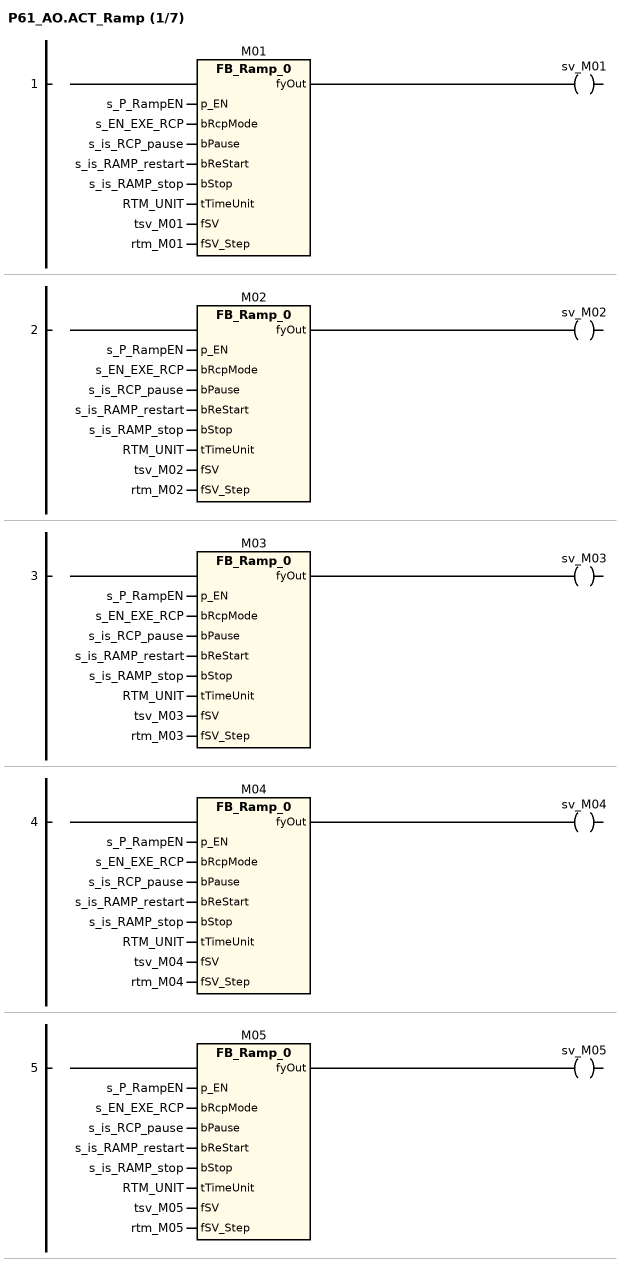
// NETWORK 1
M01(
    p_EN := s_P_RampEN,
    bRcpMode := s_EN_EXE_RCP,
    bPause := s_is_RCP_pause,
    bReStart := s_is_RAMP_restart,
    bStop := s_is_RAMP_stop,
    tTimeUnit := RTM_UNIT,
    fSV := tsv_M01,
    fSV_Step := rtm_M01); // FB_Ramp_0
sv_M01 := M01.fyOut;

// NETWORK 2
M02(
    p_EN := s_P_RampEN,
    bRcpMode := s_EN_EXE_RCP,
    bPause := s_is_RCP_pause,
    bReStart := s_is_RAMP_restart,
    bStop := s_is_RAMP_stop,
    tTimeUnit := RTM_UNIT,
    fSV := tsv_M02,
    fSV_Step := rtm_M02); // FB_Ramp_0
sv_M02 := M02.fyOut;

// NETWORK 3
M03(
    p_EN := s_P_RampEN,
    bRcpMode := s_EN_EXE_RCP,
    bPause := s_is_RCP_pause,
    bReStart := s_is_RAMP_restart,
    bStop := s_is_RAMP_stop,
    tTimeUnit := RTM_UNIT,
    fSV := tsv_M03,
    fSV_Step := rtm_M03); // FB_Ramp_0
sv_M03 := M03.fyOut;

// NETWORK 4
M04(
    p_EN := s_P_RampEN,
    bRcpMode := s_EN_EXE_RCP,
    bPause := s_is_RCP_pause,
    bReStart := s_is_RAMP_restart,
    bStop := s_is_RAMP_stop,
    tTimeUnit := RTM_UNIT,
    fSV := tsv_M04,
    fSV_Step := rtm_M04); // FB_Ramp_0
sv_M04 := M04.fyOut;

// NETWORK 5
M05(
    p_EN := s_P_RampEN,
    bRcpMode := s_EN_EXE_RCP,
    bPause := s_is_RCP_pause,
    bReStart := s_is_RAMP_restart,
    bStop := s_is_RAMP_stop,
    tTimeUnit := RTM_UNIT,
    fSV := tsv_M05,
    fSV_Step := rtm_M05); // FB_Ramp_0
sv_M05 := M05.fyOut;

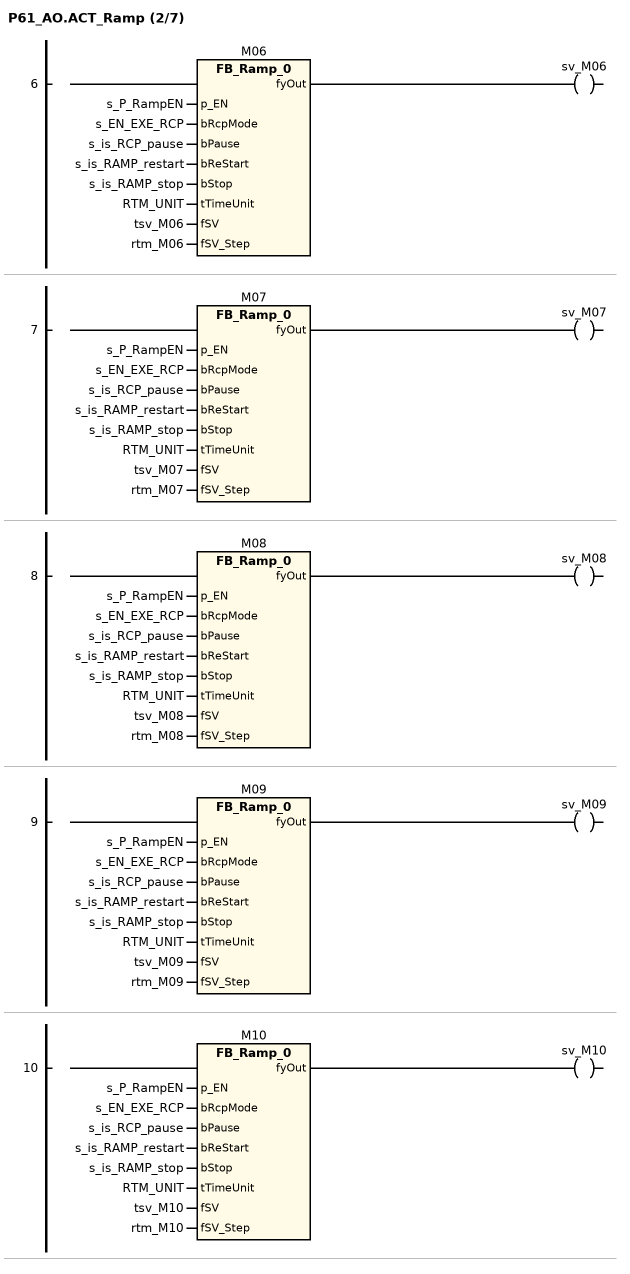
// NETWORK 6
M06(
    p_EN := s_P_RampEN,
    bRcpMode := s_EN_EXE_RCP,
    bPause := s_is_RCP_pause,
    bReStart := s_is_RAMP_restart,
    bStop := s_is_RAMP_stop,
    tTimeUnit := RTM_UNIT,
    fSV := tsv_M06,
    fSV_Step := rtm_M06); // FB_Ramp_0
sv_M06 := M06.fyOut;

// NETWORK 7
M07(
    p_EN := s_P_RampEN,
    bRcpMode := s_EN_EXE_RCP,
    bPause := s_is_RCP_pause,
    bReStart := s_is_RAMP_restart,
    bStop := s_is_RAMP_stop,
    tTimeUnit := RTM_UNIT,
    fSV := tsv_M07,
    fSV_Step := rtm_M07); // FB_Ramp_0
sv_M07 := M07.fyOut;

// NETWORK 8
M08(
    p_EN := s_P_RampEN,
    bRcpMode := s_EN_EXE_RCP,
    bPause := s_is_RCP_pause,
    bReStart := s_is_RAMP_restart,
    bStop := s_is_RAMP_stop,
    tTimeUnit := RTM_UNIT,
    fSV := tsv_M08,
    fSV_Step := rtm_M08); // FB_Ramp_0
sv_M08 := M08.fyOut;

// NETWORK 9
M09(
    p_EN := s_P_RampEN,
    bRcpMode := s_EN_EXE_RCP,
    bPause := s_is_RCP_pause,
    bReStart := s_is_RAMP_restart,
    bStop := s_is_RAMP_stop,
    tTimeUnit := RTM_UNIT,
    fSV := tsv_M09,
    fSV_Step := rtm_M09); // FB_Ramp_0
sv_M09 := M09.fyOut;

// NETWORK 10
M10(
    p_EN := s_P_RampEN,
    bRcpMode := s_EN_EXE_RCP,
    bPause := s_is_RCP_pause,
    bReStart := s_is_RAMP_restart,
    bStop := s_is_RAMP_stop,
    tTimeUnit := RTM_UNIT,
    fSV := tsv_M10,
    fSV_Step := rtm_M10); // FB_Ramp_0
sv_M10 := M10.fyOut;

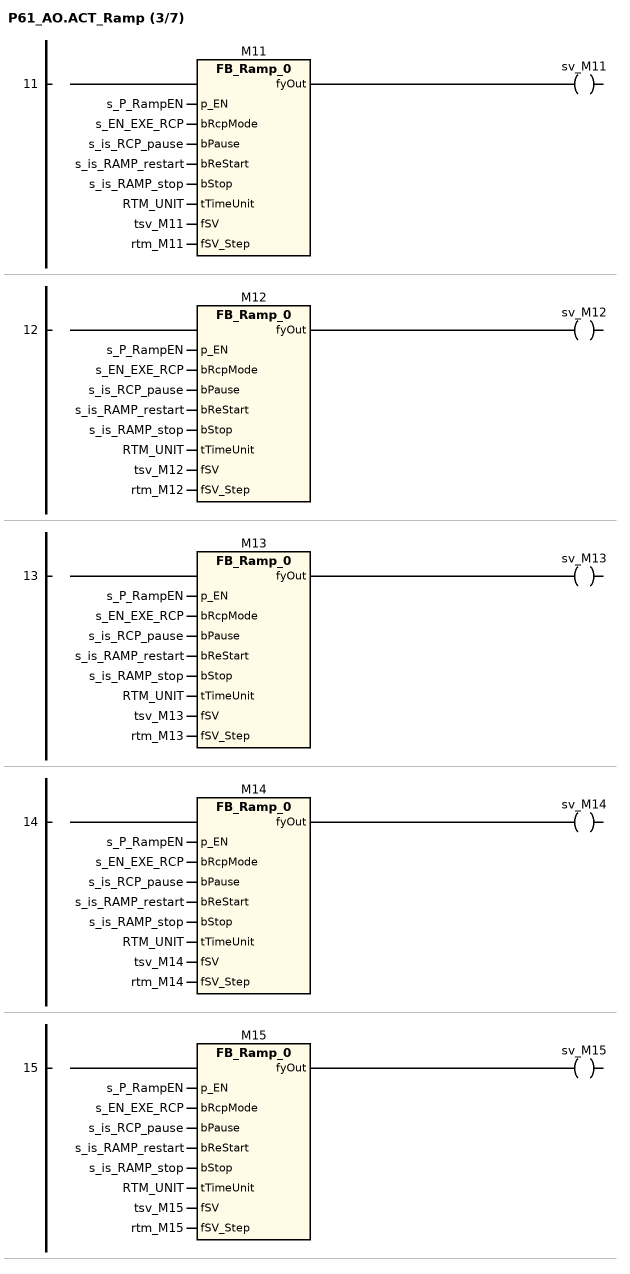
// NETWORK 11
M11(
    p_EN := s_P_RampEN,
    bRcpMode := s_EN_EXE_RCP,
    bPause := s_is_RCP_pause,
    bReStart := s_is_RAMP_restart,
    bStop := s_is_RAMP_stop,
    tTimeUnit := RTM_UNIT,
    fSV := tsv_M11,
    fSV_Step := rtm_M11); // FB_Ramp_0
sv_M11 := M11.fyOut;

// NETWORK 12
M12(
    p_EN := s_P_RampEN,
    bRcpMode := s_EN_EXE_RCP,
    bPause := s_is_RCP_pause,
    bReStart := s_is_RAMP_restart,
    bStop := s_is_RAMP_stop,
    tTimeUnit := RTM_UNIT,
    fSV := tsv_M12,
    fSV_Step := rtm_M12); // FB_Ramp_0
sv_M12 := M12.fyOut;

// NETWORK 13
M13(
    p_EN := s_P_RampEN,
    bRcpMode := s_EN_EXE_RCP,
    bPause := s_is_RCP_pause,
    bReStart := s_is_RAMP_restart,
    bStop := s_is_RAMP_stop,
    tTimeUnit := RTM_UNIT,
    fSV := tsv_M13,
    fSV_Step := rtm_M13); // FB_Ramp_0
sv_M13 := M13.fyOut;

// NETWORK 14
M14(
    p_EN := s_P_RampEN,
    bRcpMode := s_EN_EXE_RCP,
    bPause := s_is_RCP_pause,
    bReStart := s_is_RAMP_restart,
    bStop := s_is_RAMP_stop,
    tTimeUnit := RTM_UNIT,
    fSV := tsv_M14,
    fSV_Step := rtm_M14); // FB_Ramp_0
sv_M14 := M14.fyOut;

// NETWORK 15
M15(
    p_EN := s_P_RampEN,
    bRcpMode := s_EN_EXE_RCP,
    bPause := s_is_RCP_pause,
    bReStart := s_is_RAMP_restart,
    bStop := s_is_RAMP_stop,
    tTimeUnit := RTM_UNIT,
    fSV := tsv_M15,
    fSV_Step := rtm_M15); // FB_Ramp_0
sv_M15 := M15.fyOut;

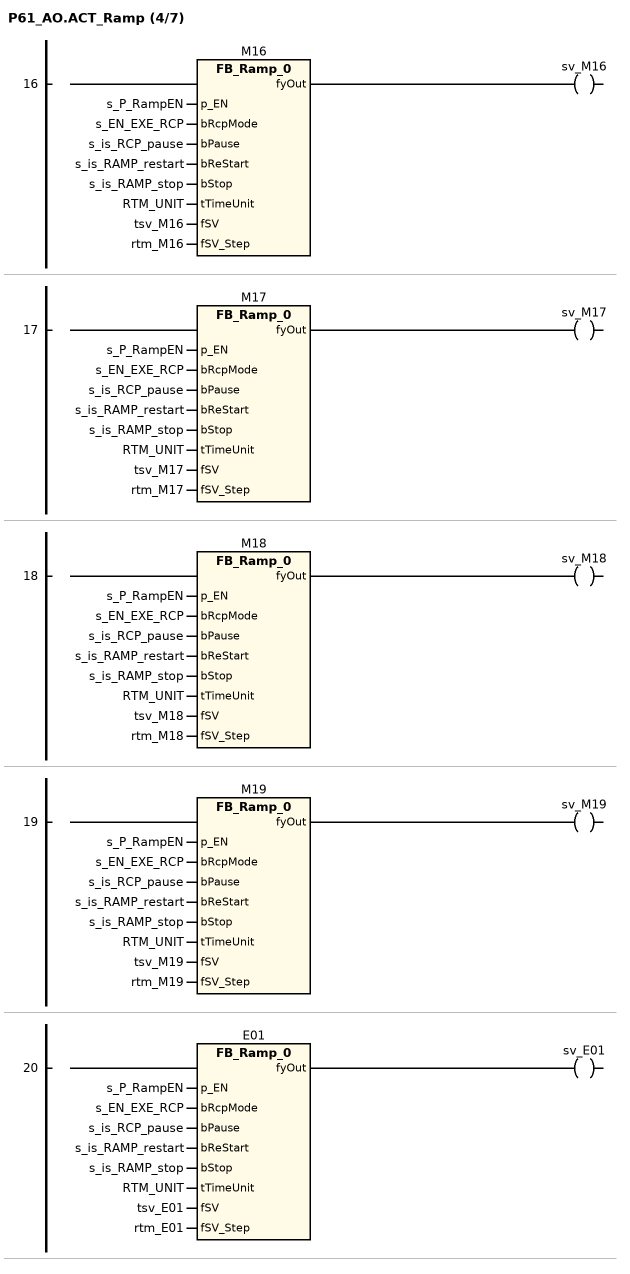
// NETWORK 16
M16(
    p_EN := s_P_RampEN,
    bRcpMode := s_EN_EXE_RCP,
    bPause := s_is_RCP_pause,
    bReStart := s_is_RAMP_restart,
    bStop := s_is_RAMP_stop,
    tTimeUnit := RTM_UNIT,
    fSV := tsv_M16,
    fSV_Step := rtm_M16); // FB_Ramp_0
sv_M16 := M16.fyOut;

// NETWORK 17
M17(
    p_EN := s_P_RampEN,
    bRcpMode := s_EN_EXE_RCP,
    bPause := s_is_RCP_pause,
    bReStart := s_is_RAMP_restart,
    bStop := s_is_RAMP_stop,
    tTimeUnit := RTM_UNIT,
    fSV := tsv_M17,
    fSV_Step := rtm_M17); // FB_Ramp_0
sv_M17 := M17.fyOut;

// NETWORK 18
M18(
    p_EN := s_P_RampEN,
    bRcpMode := s_EN_EXE_RCP,
    bPause := s_is_RCP_pause,
    bReStart := s_is_RAMP_restart,
    bStop := s_is_RAMP_stop,
    tTimeUnit := RTM_UNIT,
    fSV := tsv_M18,
    fSV_Step := rtm_M18); // FB_Ramp_0
sv_M18 := M18.fyOut;

// NETWORK 19
M19(
    p_EN := s_P_RampEN,
    bRcpMode := s_EN_EXE_RCP,
    bPause := s_is_RCP_pause,
    bReStart := s_is_RAMP_restart,
    bStop := s_is_RAMP_stop,
    tTimeUnit := RTM_UNIT,
    fSV := tsv_M19,
    fSV_Step := rtm_M19); // FB_Ramp_0
sv_M19 := M19.fyOut;

// NETWORK 20
E01(
    p_EN := s_P_RampEN,
    bRcpMode := s_EN_EXE_RCP,
    bPause := s_is_RCP_pause,
    bReStart := s_is_RAMP_restart,
    bStop := s_is_RAMP_stop,
    tTimeUnit := RTM_UNIT,
    fSV := tsv_E01,
    fSV_Step := rtm_E01); // FB_Ramp_0
sv_E01 := E01.fyOut;

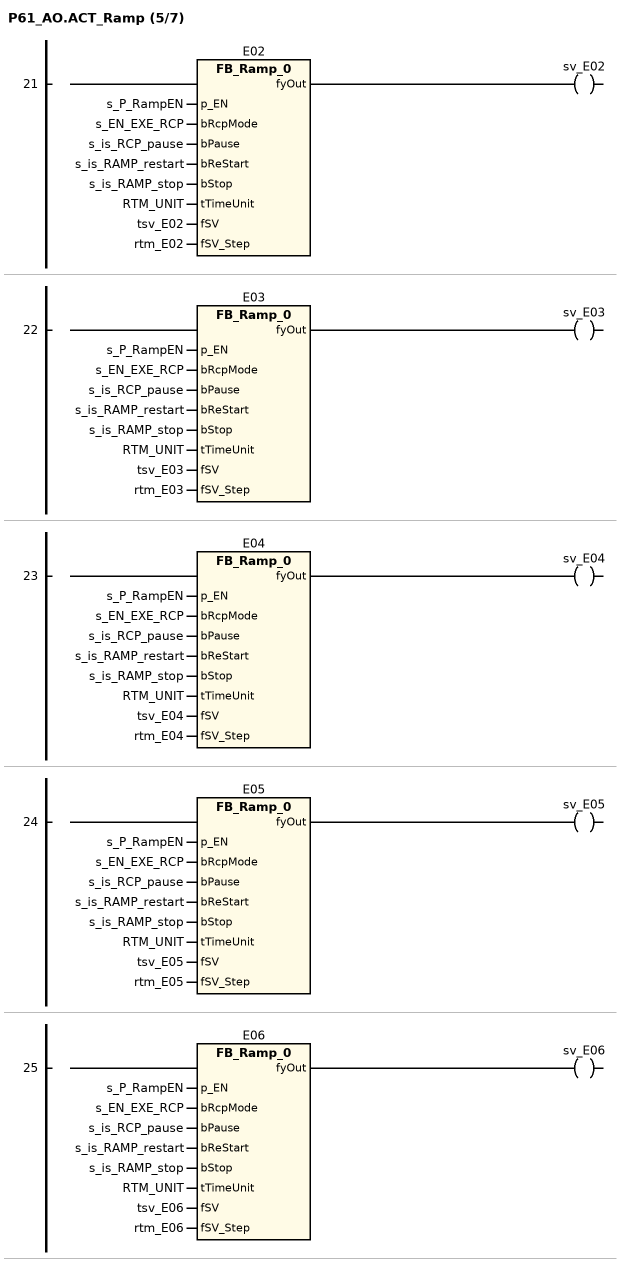
// NETWORK 21
E02(
    p_EN := s_P_RampEN,
    bRcpMode := s_EN_EXE_RCP,
    bPause := s_is_RCP_pause,
    bReStart := s_is_RAMP_restart,
    bStop := s_is_RAMP_stop,
    tTimeUnit := RTM_UNIT,
    fSV := tsv_E02,
    fSV_Step := rtm_E02); // FB_Ramp_0
sv_E02 := E02.fyOut;

// NETWORK 22
E03(
    p_EN := s_P_RampEN,
    bRcpMode := s_EN_EXE_RCP,
    bPause := s_is_RCP_pause,
    bReStart := s_is_RAMP_restart,
    bStop := s_is_RAMP_stop,
    tTimeUnit := RTM_UNIT,
    fSV := tsv_E03,
    fSV_Step := rtm_E03); // FB_Ramp_0
sv_E03 := E03.fyOut;

// NETWORK 23
E04(
    p_EN := s_P_RampEN,
    bRcpMode := s_EN_EXE_RCP,
    bPause := s_is_RCP_pause,
    bReStart := s_is_RAMP_restart,
    bStop := s_is_RAMP_stop,
    tTimeUnit := RTM_UNIT,
    fSV := tsv_E04,
    fSV_Step := rtm_E04); // FB_Ramp_0
sv_E04 := E04.fyOut;

// NETWORK 24
E05(
    p_EN := s_P_RampEN,
    bRcpMode := s_EN_EXE_RCP,
    bPause := s_is_RCP_pause,
    bReStart := s_is_RAMP_restart,
    bStop := s_is_RAMP_stop,
    tTimeUnit := RTM_UNIT,
    fSV := tsv_E05,
    fSV_Step := rtm_E05); // FB_Ramp_0
sv_E05 := E05.fyOut;

// NETWORK 25
E06(
    p_EN := s_P_RampEN,
    bRcpMode := s_EN_EXE_RCP,
    bPause := s_is_RCP_pause,
    bReStart := s_is_RAMP_restart,
    bStop := s_is_RAMP_stop,
    tTimeUnit := RTM_UNIT,
    fSV := tsv_E06,
    fSV_Step := rtm_E06); // FB_Ramp_0
sv_E06 := E06.fyOut;

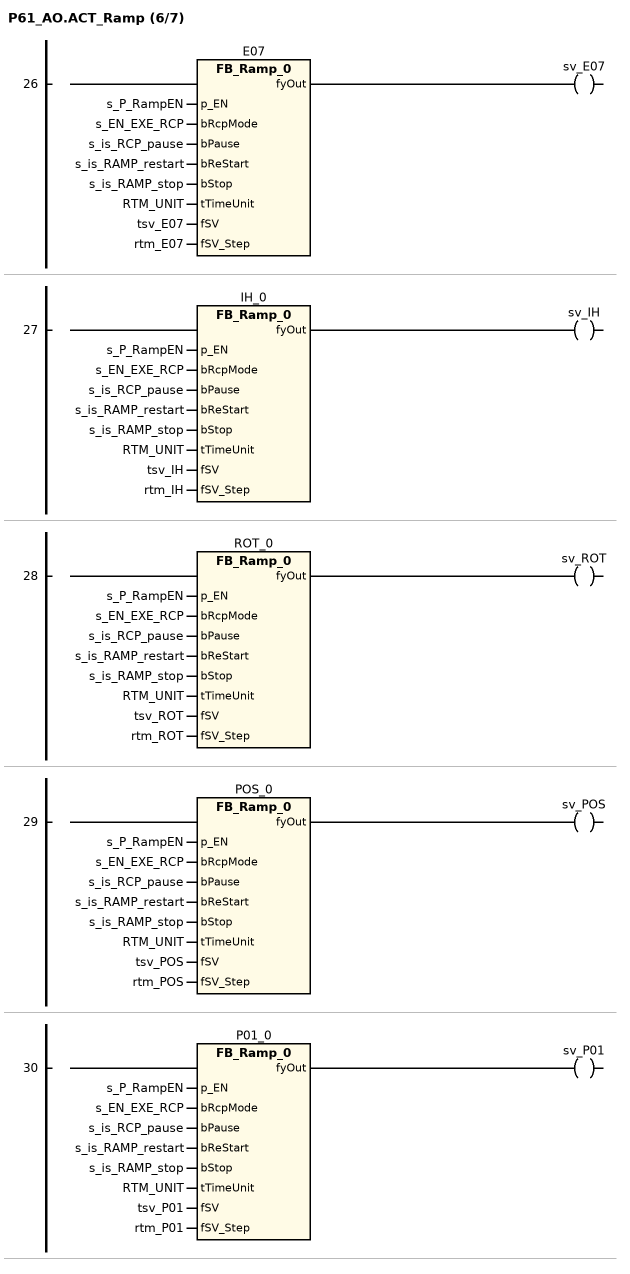
// NETWORK 26
E07(
    p_EN := s_P_RampEN,
    bRcpMode := s_EN_EXE_RCP,
    bPause := s_is_RCP_pause,
    bReStart := s_is_RAMP_restart,
    bStop := s_is_RAMP_stop,
    tTimeUnit := RTM_UNIT,
    fSV := tsv_E07,
    fSV_Step := rtm_E07); // FB_Ramp_0
sv_E07 := E07.fyOut;

// NETWORK 27
IH_0(
    p_EN := s_P_RampEN,
    bRcpMode := s_EN_EXE_RCP,
    bPause := s_is_RCP_pause,
    bReStart := s_is_RAMP_restart,
    bStop := s_is_RAMP_stop,
    tTimeUnit := RTM_UNIT,
    fSV := tsv_IH,
    fSV_Step := rtm_IH); // FB_Ramp_0
sv_IH := IH_0.fyOut;

// NETWORK 28
ROT_0(
    p_EN := s_P_RampEN,
    bRcpMode := s_EN_EXE_RCP,
    bPause := s_is_RCP_pause,
    bReStart := s_is_RAMP_restart,
    bStop := s_is_RAMP_stop,
    tTimeUnit := RTM_UNIT,
    fSV := tsv_ROT,
    fSV_Step := rtm_ROT); // FB_Ramp_0
sv_ROT := ROT_0.fyOut;

// NETWORK 29
POS_0(
    p_EN := s_P_RampEN,
    bRcpMode := s_EN_EXE_RCP,
    bPause := s_is_RCP_pause,
    bReStart := s_is_RAMP_restart,
    bStop := s_is_RAMP_stop,
    tTimeUnit := RTM_UNIT,
    fSV := tsv_POS,
    fSV_Step := rtm_POS); // FB_Ramp_0
sv_POS := POS_0.fyOut;

// NETWORK 30
P01_0(
    p_EN := s_P_RampEN,
    bRcpMode := s_EN_EXE_RCP,
    bPause := s_is_RCP_pause,
    bReStart := s_is_RAMP_restart,
    bStop := s_is_RAMP_stop,
    tTimeUnit := RTM_UNIT,
    fSV := tsv_P01,
    fSV_Step := rtm_P01); // FB_Ramp_0
sv_P01 := P01_0.fyOut;

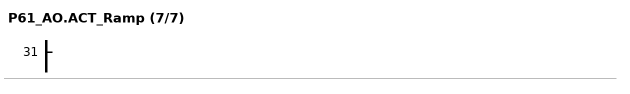
// NETWORK 31
END_ACTION

ACTION ACT_Ramp_OLD:
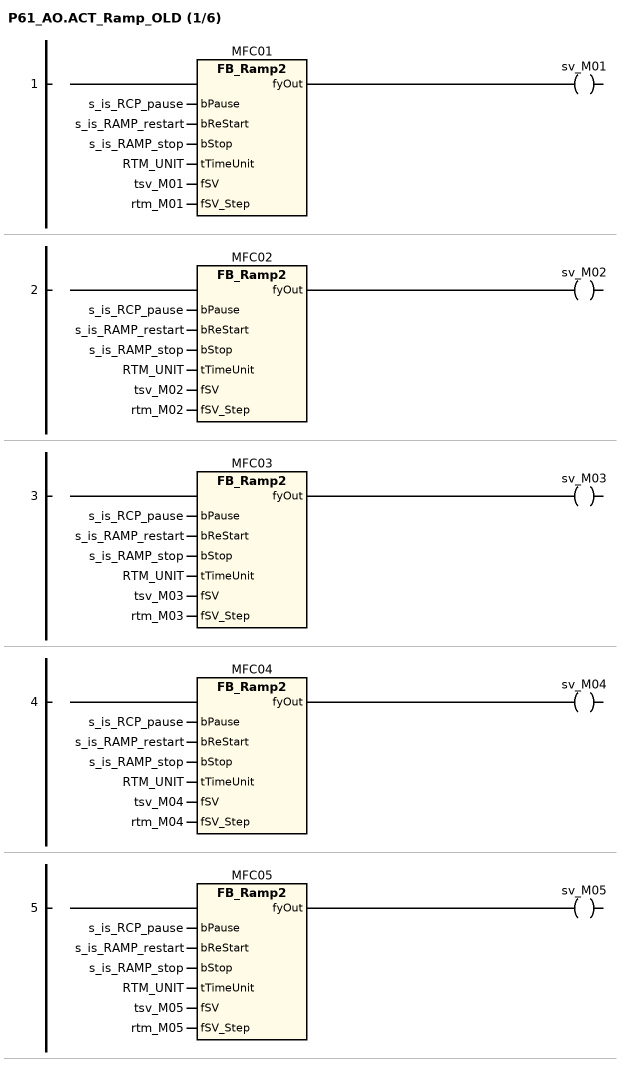
// NETWORK 1
MFC01(
    bPause := s_is_RCP_pause,
    bReStart := s_is_RAMP_restart,
    bStop := s_is_RAMP_stop,
    tTimeUnit := RTM_UNIT,
    fSV := tsv_M01,
    fSV_Step := rtm_M01); // FB_Ramp2
sv_M01 := MFC01.fyOut;

// NETWORK 2
MFC02(
    bPause := s_is_RCP_pause,
    bReStart := s_is_RAMP_restart,
    bStop := s_is_RAMP_stop,
    tTimeUnit := RTM_UNIT,
    fSV := tsv_M02,
    fSV_Step := rtm_M02); // FB_Ramp2
sv_M02 := MFC02.fyOut;

// NETWORK 3
MFC03(
    bPause := s_is_RCP_pause,
    bReStart := s_is_RAMP_restart,
    bStop := s_is_RAMP_stop,
    tTimeUnit := RTM_UNIT,
    fSV := tsv_M03,
    fSV_Step := rtm_M03); // FB_Ramp2
sv_M03 := MFC03.fyOut;

// NETWORK 4
MFC04(
    bPause := s_is_RCP_pause,
    bReStart := s_is_RAMP_restart,
    bStop := s_is_RAMP_stop,
    tTimeUnit := RTM_UNIT,
    fSV := tsv_M04,
    fSV_Step := rtm_M04); // FB_Ramp2
sv_M04 := MFC04.fyOut;

// NETWORK 5
MFC05(
    bPause := s_is_RCP_pause,
    bReStart := s_is_RAMP_restart,
    bStop := s_is_RAMP_stop,
    tTimeUnit := RTM_UNIT,
    fSV := tsv_M05,
    fSV_Step := rtm_M05); // FB_Ramp2
sv_M05 := MFC05.fyOut;

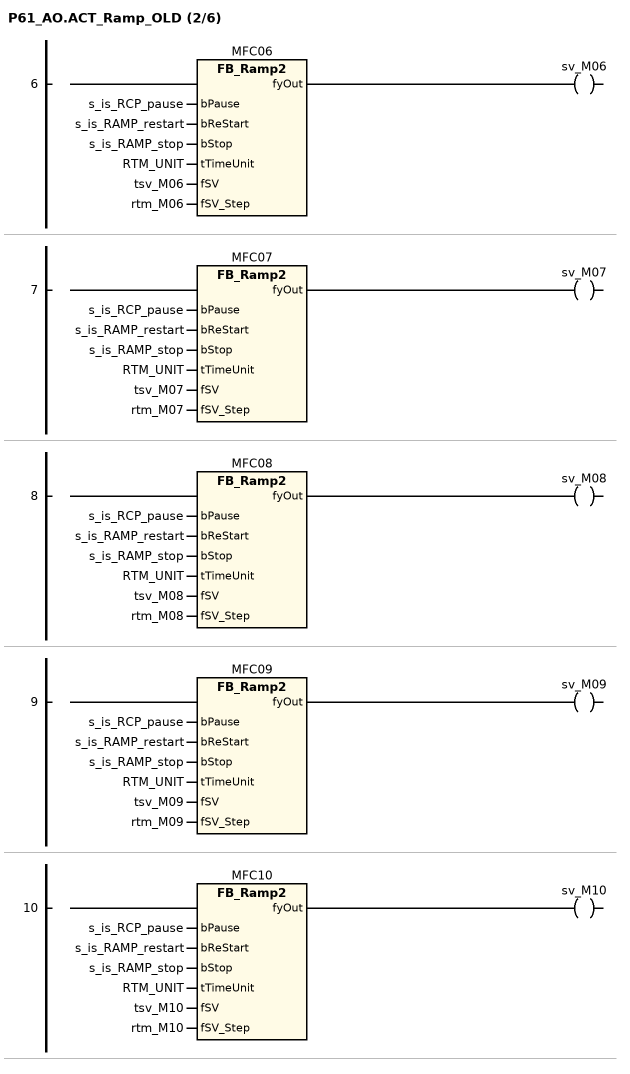
// NETWORK 6
MFC06(
    bPause := s_is_RCP_pause,
    bReStart := s_is_RAMP_restart,
    bStop := s_is_RAMP_stop,
    tTimeUnit := RTM_UNIT,
    fSV := tsv_M06,
    fSV_Step := rtm_M06); // FB_Ramp2
sv_M06 := MFC06.fyOut;

// NETWORK 7
MFC07(
    bPause := s_is_RCP_pause,
    bReStart := s_is_RAMP_restart,
    bStop := s_is_RAMP_stop,
    tTimeUnit := RTM_UNIT,
    fSV := tsv_M07,
    fSV_Step := rtm_M07); // FB_Ramp2
sv_M07 := MFC07.fyOut;

// NETWORK 8
MFC08(
    bPause := s_is_RCP_pause,
    bReStart := s_is_RAMP_restart,
    bStop := s_is_RAMP_stop,
    tTimeUnit := RTM_UNIT,
    fSV := tsv_M08,
    fSV_Step := rtm_M08); // FB_Ramp2
sv_M08 := MFC08.fyOut;

// NETWORK 9
MFC09(
    bPause := s_is_RCP_pause,
    bReStart := s_is_RAMP_restart,
    bStop := s_is_RAMP_stop,
    tTimeUnit := RTM_UNIT,
    fSV := tsv_M09,
    fSV_Step := rtm_M09); // FB_Ramp2
sv_M09 := MFC09.fyOut;

// NETWORK 10
MFC10(
    bPause := s_is_RCP_pause,
    bReStart := s_is_RAMP_restart,
    bStop := s_is_RAMP_stop,
    tTimeUnit := RTM_UNIT,
    fSV := tsv_M10,
    fSV_Step := rtm_M10); // FB_Ramp2
sv_M10 := MFC10.fyOut;

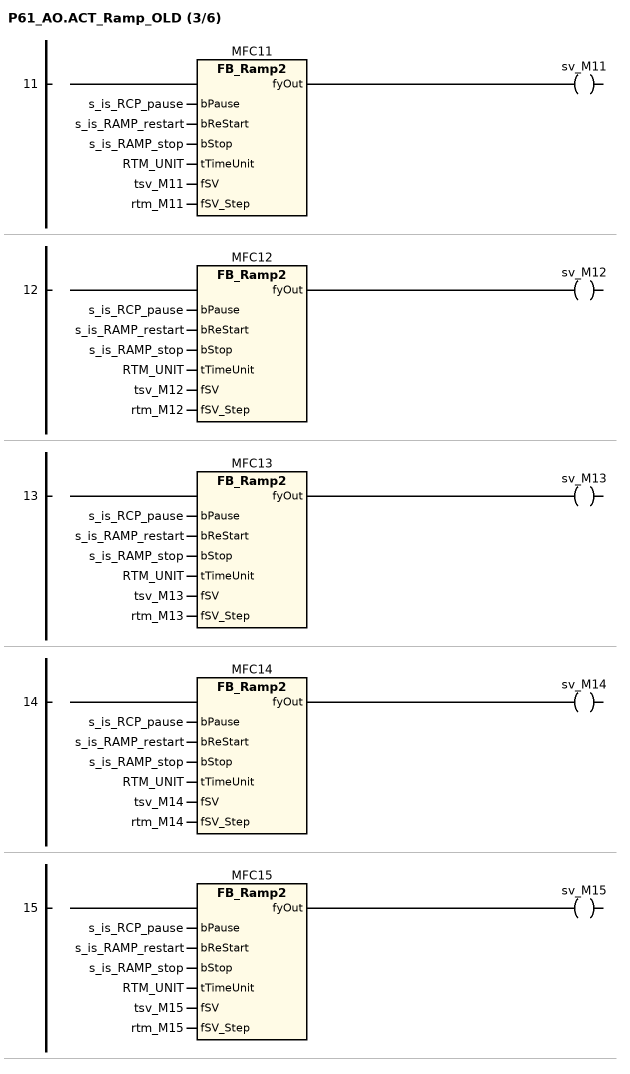
// NETWORK 11
MFC11(
    bPause := s_is_RCP_pause,
    bReStart := s_is_RAMP_restart,
    bStop := s_is_RAMP_stop,
    tTimeUnit := RTM_UNIT,
    fSV := tsv_M11,
    fSV_Step := rtm_M11); // FB_Ramp2
sv_M11 := MFC11.fyOut;

// NETWORK 12
MFC12(
    bPause := s_is_RCP_pause,
    bReStart := s_is_RAMP_restart,
    bStop := s_is_RAMP_stop,
    tTimeUnit := RTM_UNIT,
    fSV := tsv_M12,
    fSV_Step := rtm_M12); // FB_Ramp2
sv_M12 := MFC12.fyOut;

// NETWORK 13
MFC13(
    bPause := s_is_RCP_pause,
    bReStart := s_is_RAMP_restart,
    bStop := s_is_RAMP_stop,
    tTimeUnit := RTM_UNIT,
    fSV := tsv_M13,
    fSV_Step := rtm_M13); // FB_Ramp2
sv_M13 := MFC13.fyOut;

// NETWORK 14
MFC14(
    bPause := s_is_RCP_pause,
    bReStart := s_is_RAMP_restart,
    bStop := s_is_RAMP_stop,
    tTimeUnit := RTM_UNIT,
    fSV := tsv_M14,
    fSV_Step := rtm_M14); // FB_Ramp2
sv_M14 := MFC14.fyOut;

// NETWORK 15
MFC15(
    bPause := s_is_RCP_pause,
    bReStart := s_is_RAMP_restart,
    bStop := s_is_RAMP_stop,
    tTimeUnit := RTM_UNIT,
    fSV := tsv_M15,
    fSV_Step := rtm_M15); // FB_Ramp2
sv_M15 := MFC15.fyOut;

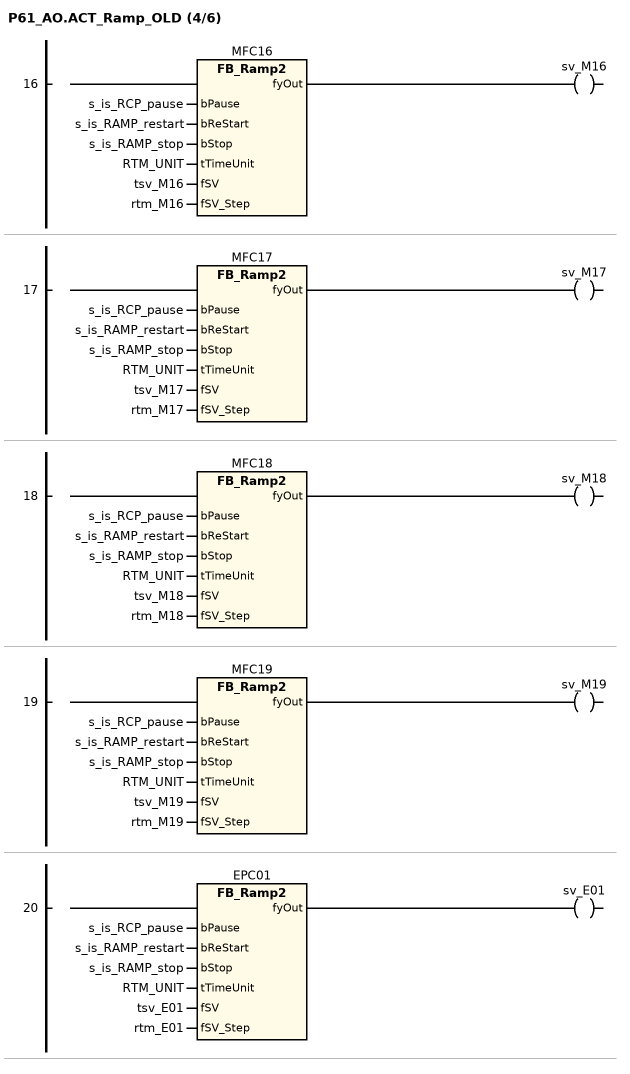
// NETWORK 16
MFC16(
    bPause := s_is_RCP_pause,
    bReStart := s_is_RAMP_restart,
    bStop := s_is_RAMP_stop,
    tTimeUnit := RTM_UNIT,
    fSV := tsv_M16,
    fSV_Step := rtm_M16); // FB_Ramp2
sv_M16 := MFC16.fyOut;

// NETWORK 17
MFC17(
    bPause := s_is_RCP_pause,
    bReStart := s_is_RAMP_restart,
    bStop := s_is_RAMP_stop,
    tTimeUnit := RTM_UNIT,
    fSV := tsv_M17,
    fSV_Step := rtm_M17); // FB_Ramp2
sv_M17 := MFC17.fyOut;

// NETWORK 18
MFC18(
    bPause := s_is_RCP_pause,
    bReStart := s_is_RAMP_restart,
    bStop := s_is_RAMP_stop,
    tTimeUnit := RTM_UNIT,
    fSV := tsv_M18,
    fSV_Step := rtm_M18); // FB_Ramp2
sv_M18 := MFC18.fyOut;

// NETWORK 19
MFC19(
    bPause := s_is_RCP_pause,
    bReStart := s_is_RAMP_restart,
    bStop := s_is_RAMP_stop,
    tTimeUnit := RTM_UNIT,
    fSV := tsv_M19,
    fSV_Step := rtm_M19); // FB_Ramp2
sv_M19 := MFC19.fyOut;

// NETWORK 20
EPC01(
    bPause := s_is_RCP_pause,
    bReStart := s_is_RAMP_restart,
    bStop := s_is_RAMP_stop,
    tTimeUnit := RTM_UNIT,
    fSV := tsv_E01,
    fSV_Step := rtm_E01); // FB_Ramp2
sv_E01 := EPC01.fyOut;

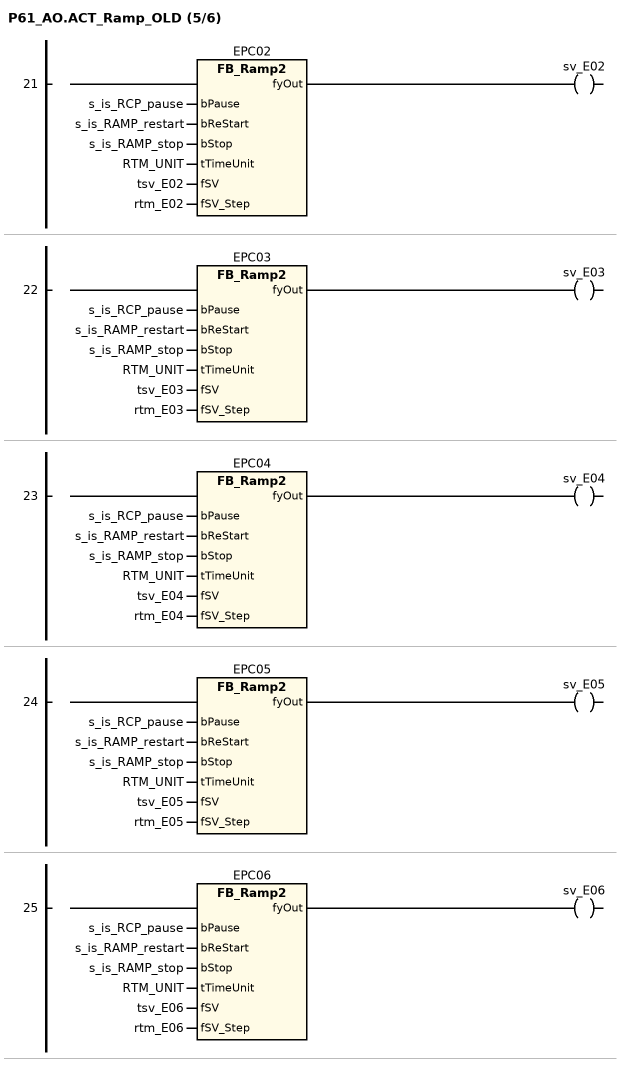
// NETWORK 21
EPC02(
    bPause := s_is_RCP_pause,
    bReStart := s_is_RAMP_restart,
    bStop := s_is_RAMP_stop,
    tTimeUnit := RTM_UNIT,
    fSV := tsv_E02,
    fSV_Step := rtm_E02); // FB_Ramp2
sv_E02 := EPC02.fyOut;

// NETWORK 22
EPC03(
    bPause := s_is_RCP_pause,
    bReStart := s_is_RAMP_restart,
    bStop := s_is_RAMP_stop,
    tTimeUnit := RTM_UNIT,
    fSV := tsv_E03,
    fSV_Step := rtm_E03); // FB_Ramp2
sv_E03 := EPC03.fyOut;

// NETWORK 23
EPC04(
    bPause := s_is_RCP_pause,
    bReStart := s_is_RAMP_restart,
    bStop := s_is_RAMP_stop,
    tTimeUnit := RTM_UNIT,
    fSV := tsv_E04,
    fSV_Step := rtm_E04); // FB_Ramp2
sv_E04 := EPC04.fyOut;

// NETWORK 24
EPC05(
    bPause := s_is_RCP_pause,
    bReStart := s_is_RAMP_restart,
    bStop := s_is_RAMP_stop,
    tTimeUnit := RTM_UNIT,
    fSV := tsv_E05,
    fSV_Step := rtm_E05); // FB_Ramp2
sv_E05 := EPC05.fyOut;

// NETWORK 25
EPC06(
    bPause := s_is_RCP_pause,
    bReStart := s_is_RAMP_restart,
    bStop := s_is_RAMP_stop,
    tTimeUnit := RTM_UNIT,
    fSV := tsv_E06,
    fSV_Step := rtm_E06); // FB_Ramp2
sv_E06 := EPC06.fyOut;

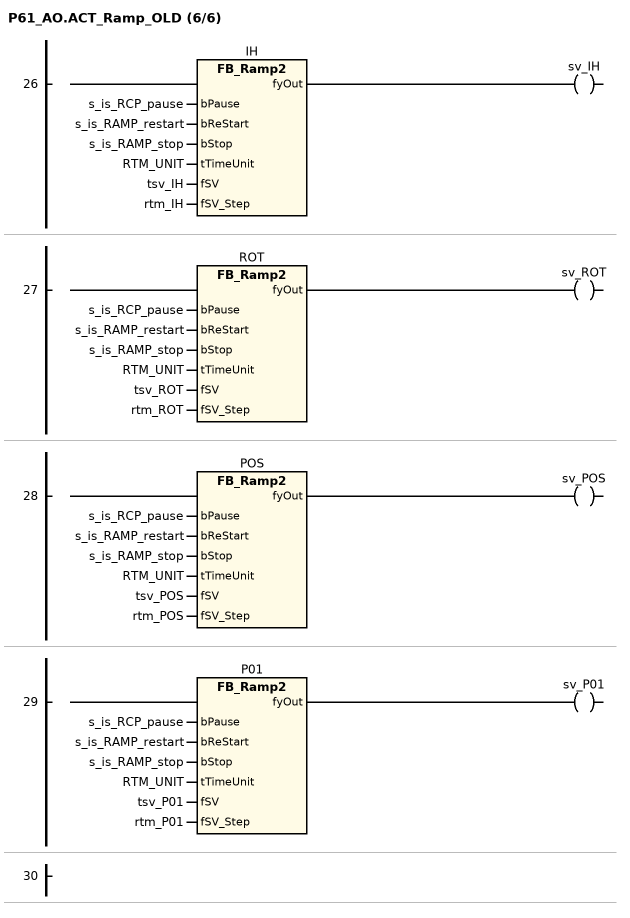
// NETWORK 26
IH(
    bPause := s_is_RCP_pause,
    bReStart := s_is_RAMP_restart,
    bStop := s_is_RAMP_stop,
    tTimeUnit := RTM_UNIT,
    fSV := tsv_IH,
    fSV_Step := rtm_IH); // FB_Ramp2
sv_IH := IH.fyOut;

// NETWORK 27
ROT(
    bPause := s_is_RCP_pause,
    bReStart := s_is_RAMP_restart,
    bStop := s_is_RAMP_stop,
    tTimeUnit := RTM_UNIT,
    fSV := tsv_ROT,
    fSV_Step := rtm_ROT); // FB_Ramp2
sv_ROT := ROT.fyOut;

// NETWORK 28
POS(
    bPause := s_is_RCP_pause,
    bReStart := s_is_RAMP_restart,
    bStop := s_is_RAMP_stop,
    tTimeUnit := RTM_UNIT,
    fSV := tsv_POS,
    fSV_Step := rtm_POS); // FB_Ramp2
sv_POS := POS.fyOut;

// NETWORK 29
P01(
    bPause := s_is_RCP_pause,
    bReStart := s_is_RAMP_restart,
    bStop := s_is_RAMP_stop,
    tTimeUnit := RTM_UNIT,
    fSV := tsv_P01,
    fSV_Step := rtm_P01); // FB_Ramp2
sv_P01 := P01.fyOut;

// NETWORK 30
END_ACTION

END_PROGRAM

// ---- POUs/MR_PRG/REF_P02_KL1501.TcPOU
PROGRAM REF_P02_KL1501
VAR
	//bError: BOOL;
	t_1S: TON;	
	
	iStatus: USINT;
	in1: UINT;
	in2: UINT;
		
	encCount: UDINT;
	inData: ST_KL1501InData;
	outData: ST_KL1501OutData;
	KL1501Cfg: FB_KL1501Config;
	
	One_Turn_PLS: REAL ;
	PLS_Old: REAL := 0;
	PLS_New: REAL := 0;
	PLS_Diff: REAL := 0;
	Encoder_Max: REAL := 4294967295; //UINT Range 0 ~ 65,535
	RPM_PV: REAL := 0;
	FB_RPM_AVG: FB_AVG10;
	RPM_AVG: REAL;
    BLDC_MAX_RPM_PLS: REAL := 36000;//genicom : 12PULSE * 3000RPM = 36,000PULSE, china hvpe :500PULSE * 4000RPM = 2,000,000PULSE	
END_VAR

t_1S(PT := T#1S);
t_1S.IN := ON;

//KL1501 Not Use
(*

inData.iState := XA_ENC_ST;
inData.arrDataIn[0] := XA_ENC_IN[0];
inData.arrDataIn[1] := XA_ENC_IN[1];

IF t_1S.Q THEN
	t_1S.IN := Off;
	
	ACT_KL1501();
	
	//Rotation - BLDC Encoder
	pv_ENC := PLS_New := UDINT_TO_REAL(encCount);
	IF N_MAX[29] > 0 THEN
		One_Turn_PLS := BLDC_MAX_RPM_PLS / N_MAX[29];
	ELSE
		One_Turn_PLS := 1;
	END_IF
	IF PLS_New <> PLS_Old THEN //pulse input check
		IF PLS_New <= PLS_Old THEN//Ring counter Check
			PLS_New := PLS_New + Encoder_Max;
		END_IF
		PLS_Diff := PLS_New - PLS_Old;//PLS_Diff is always + value	
		IF PLS_Diff >= 0 THEN	//PLS_Diff is sometime abnormal value
			pv_ROT_inchPulse := pv_ROT_inchPulse + PLS_Diff; //PLS_Diff is always + value
			pv_ROT_1turnPulse := pv_ROT_1turnPulse + PLS_Diff; //PLS_Diff is always + value
			RPM_PV := PLS_Diff * 60 / One_Turn_PLS ;// 60 = 60Sec
		END_IF
		pv_ROT := RPM_PV;
	ELSE	
		pv_ROT := 0;	
	END_IF
	
	IF pv_ROT_1turnPulse >= One_Turn_PLS THEN
		pv_ROT_1turnPulse := pv_ROT_1turnPulse - One_Turn_PLS;
	END_IF
	pv_ROT_DEGREE := pv_ROT_1turnPulse *  360 / One_Turn_PLS;
	
	is_ROT_plsActived := PLS_New <> PLS_Old;
	PLS_Old := PLS_New;	

END_IF;//end 1Sec Timer.Q

*)

ACTION ACT_KL1501:
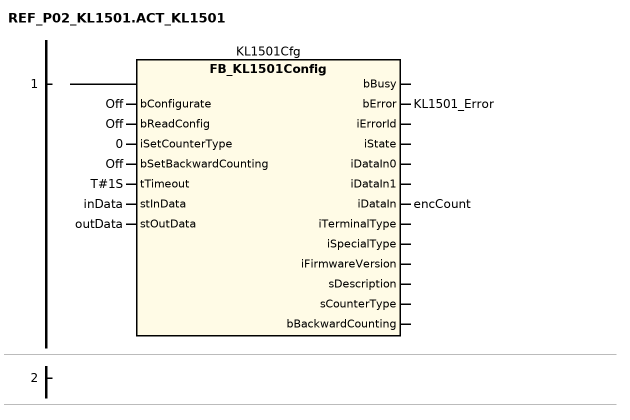
// NETWORK 1
KL1501Cfg(
    bConfigurate := Off,
    bReadConfig := Off,
    iSetCounterType := 0,
    bSetBackwardCounting := Off,
    tTimeout := T#1S,
    stInData := inData,
    stOutData := outData,
    bError => KL1501_Error,
    iDataIn => encCount); // FB_KL1501Config

// NETWORK 2
END_ACTION

END_PROGRAM

// ---- POUs/P02_P2P/P00_Task_Fast.TcPOU
PROGRAM P00_Task_Fast
VAR
END_VAR


Task_Fast_LH();
Task_Fast_TB();

END_PROGRAM

// ---- POUs/P02_P2P/Task_Fast_LH.TcPOU
PROGRAM Task_Fast_LH
VAR
	//LineHeater Controller(MC9-8RD0SS32) x 1EA
	(* background communication with the KL6031 terminal (22byte) *)
	fbCtrl: SerialLineControl;
	bCtrlError: BOOL;
	eCtrlErrorID: ComError_t;
	fbKLConfig: KL6configuration;
	bKLConfigError: BOOL;
	eKLConfigErrorID: ComError_t;
	bKLConfigExe: BOOL := TRUE;
END_VAR

//LH: Line Heater x 8EA -> 8Channel TIC 1EA
//Maker: HANYOUNG NUX
//Model: MC9-8RD0SS32
//Temp Range: -15 ~200℃
//RS485: 9600, DataBit(8), Parity(None), StopBit(1)
//BCC Check X
fbCtrl(
	Mode:= SERIALLINEMODE_KL6_22B_STANDARD,
	pComIn:= ADR(in22B_LH),
	pComOut:= ADR(out22B_LH),
	SizeComIn:= SIZEOF(in22B_LH),
	Error=> ,
	ErrorID=> ,
	TxBuffer:= TxBuf_LH,
	RxBuffer:= RxBuf_LH );
IF fbCtrl.Error THEN
	bCtrlError := TRUE;
	eCtrlErrorID := fbCtrl.ErrorID;
END_IF

END_PROGRAM

// ---- POUs/P02_P2P/Task_Fast_TB.TcPOU
PROGRAM Task_Fast_TB
VAR
	//Thermal Bath(HEBC002-WA10) x 6EA
	(* background communication with the KL6031 terminal (22byte) *)
	fbCtrl: SerialLineControl;
	bCtrlError: BOOL;
	eCtrlErrorID: ComError_t;
	fbKLConfig: KL6configuration;
	bKLConfigError: BOOL;
	eKLConfigErrorID: ComError_t;
	bKLConfigExe: BOOL := TRUE;	
END_VAR

//TB: Thermal Bath x 6EA
//Maker: SMC
//Model: HEBC002-WA10
//Temp Range: -15 ~60℃
//RS485: 9600, DataBit(8), Parity(None), StopBit(1)
//BCC Check X
fbCtrl(
	Mode:= SERIALLINEMODE_KL6_22B_STANDARD,
	pComIn:= ADR(in22B_TB),
	pComOut:= ADR(out22B_TB),
	SizeComIn:= SIZEOF(in22B_TB),
	Error=> ,
	ErrorID=> ,
	TxBuffer:= TxBuf_TB,
	RxBuffer:= RxBuf_TB );
IF fbCtrl.Error THEN
	bCtrlError := TRUE;
	eCtrlErrorID := fbCtrl.ErrorID;
END_IF

END_PROGRAM

// ---- POUs/TextFieldInputHandler.TcPOU
// 텍스트 필드 편집이 완료되었을 때 알림을 받기 위한 FB
// Recipe Values table에 사용됨
FUNCTION_BLOCK TextfieldInputHandler
VAR_INPUT
		finishedEdit  :BOOL; // 변수가 작성되었을 때 TRUE 설정. 
                             // 편집하기 전에 FALSE로 설정해야 유용함. write variable action이 있는 텍스트필드의 action에 수행할 수 있음.
END_VAR
VAR
END_VAR

// no implementation here since Method is where the action happens

 (*이 메서드는 시각화 사용자가 변수를 작성한 후에 호출됨. 변수는 입력필드를 사용하여 작성됨.
    이 메서드에 대한 호출은 VISU_TASK에서 수행되므로 다른 작업과 동기화가 필요한 작업을 수행할 때는 주의*)
METHOD VariableWritten : BOOL
VAR_INPUT

 (*작성된 변수에 대한 포인터. POINT TO BYTE는 사용된 변수의 구체적인 형식에 대한 placeholder로 사용됨 
   변경된 변수에 접근하려면 이 포인터를 올바른 유형 (예:포인터를 DWORD로 변경)로 캐스팅할 수 있음
   type에 대한 정보는 <see cref="varType"/>으로 볼 수 있음*)
 pVar	: POINTER TO BYTE;
	(* 작성된 변수의 형식*)
//	varType	: CmpVisuHandler.Visu_Types;
	(* bytes 사이즈로 변수의 최대 크기 (형식이 stringtype 경우에만 유효함 , 그 이외에 0보다 작음). *)
	iMaxSize	: INT;
	(* 이 값을 사용하는 client structured에 대한 포인터*)
//	pClient	: POINTER TO VisuElemBase.VisuStructClientData;
END_VAR
finishedEdit := TRUE;
END_METHOD

END_FUNCTION_BLOCK

// ---- POUs/VisuInit.TcPOU
PROGRAM VisuInit
VAR_INPUT
	TFHandler : TextfieldInputHandler;
END_VAR

//VisuElems.g_VisuEventManager.SetEditBoxEventHandler(handler := TFHandler);

END_PROGRAM
